FUNCTION_BLOCK AUI_CTU (* Event driven up counter (Adapter Version) - On Change Triggering *)
  (* Standard: 61499-1 Annex 2; Description: Copyright (c) 2017 fortiss GmbH, HR Agrartechnik GmbH This program and the accompanying materials are made available under the terms of the Eclipse Public License 2.0 which is available at https://www.eclipse.org/legal/epl-2.0/ SPDX-License-Identifier: EPL-2.0 *)
  (* Version 3.2, 2026-04-19, Franz Höpfinger, Made Q event triggering on-change only via internal state tracking *)
  (* Version 3.1, 2026-04-19, Franz Höpfinger, Added status event for Q adapter and PV update logic *)
  (* Version 3.0, 2025-04-14, Patrick Aigner, changed package *)
  (* Version 1.0, 2017-09-21, Alois Zoitl, fortiss GmbH, initial API and implementation and/or initial documentation *)
  PACKAGE adapter::events::unidirectional;
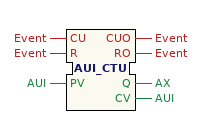
  EVENT_INPUT
    CU; (* Count up *)
    R; (* Reset *)
  END_EVENT
  EVENT_OUTPUT
    CUO; (* Count up output *)
    RO; (* Reset output *)
  END_EVENT
  SOCKETS
    PV : adapter::types::unidirectional::AUI; (* Process Value *)
  END_SOCKETS
  PLUGS
    Q : adapter::types::unidirectional::AX; (* True if CV >= PV *)
    CV : adapter::types::unidirectional::AUI; (* Counter Value *)
  END_PLUGS
  VAR
    Q_OLD : BOOL := FALSE; (* Stores the previous state of the output Q to detect changes (On-Change triggering) *) {SET_ATTRIBUTE(Retain, NON_RETAIN)}
  END_VAR
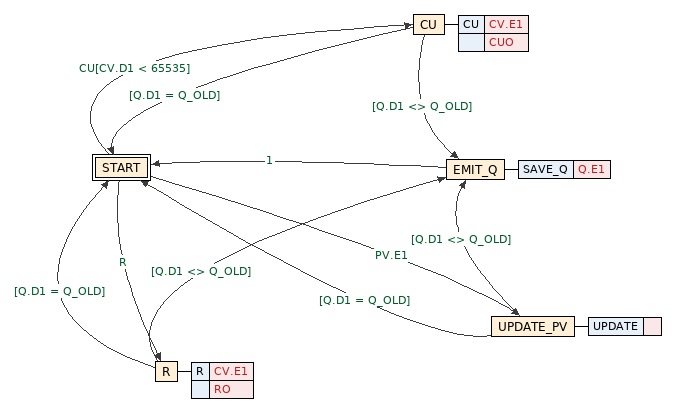
  EC_STATES
    START; (* Initial State *)
    CU : CU -> CV.E1, -> CUO; (* Count Up *)
    R : R -> CV.E1, -> RO; (* Reset *)
    UPDATE_PV : UPDATE; (* Re-evaluate Q on PV change *)
    EMIT_Q : SAVE_Q -> Q.E1; (* Fires Q event and saves state *)
  END_STATES
  EC_TRANSITIONS
    START TO CU := CU[CV.D1 < 65535];
    CU TO EMIT_Q := [Q.D1 <> Q_OLD];
    CU TO START := [Q.D1 = Q_OLD];
    START TO R := R;
    R TO EMIT_Q := [Q.D1 <> Q_OLD];
    R TO START := [Q.D1 = Q_OLD];
    START TO UPDATE_PV := PV.E1;
    UPDATE_PV TO EMIT_Q := [Q.D1 <> Q_OLD];
    UPDATE_PV TO START := [Q.D1 = Q_OLD];
    EMIT_Q TO START := 1;
  END_TRANSITIONS
  ALGORITHM R IN ST: (* reset counter *)
CV.D1 := 0;
Q.D1 := (CV.D1 >= PV.D1);
  END_ALGORITHM
  ALGORITHM CU IN ST: (* count up *)
CV.D1 := CV.D1 + 1;
Q.D1 := (CV.D1 >= PV.D1);
  END_ALGORITHM
  ALGORITHM UPDATE IN ST: (* update status only *)
Q.D1 := (CV.D1 >= PV.D1);
  END_ALGORITHM
  ALGORITHM SAVE_Q IN ST: (* save state *)
Q_OLD := Q.D1;
  END_ALGORITHM
END_FUNCTION_BLOCK
